Omron CX-Programmer project NewProject (CX-Programmer 9.73)

# PLC NewPLC1: CP1E N30

## Global symbols (name address type ; comment)
0.00 BOOL  ; START
0.01 BOOL  ; STOP
100.00 BOOL  ; LAMPU HIJAU SIMPANG 1
100.01 BOOL  ; LAMPU KUNING SIMPANG 1
100.02 BOOL  ; LAMPU MERAH SIMPANG 1
100.03 BOOL  ; LAMPU HIJAU SIMPANG 2
100.04 BOOL  ; LAMPU KUNING SIMPANG 2
100.05 BOOL  ; LAMPU MERAH SIMPANG 2
100.06 BOOL  ; LAMPU HIJAU SIMPANG 3
100.07 BOOL  ; LAMPU KUNING SIMPANG 3
100.08 BOOL  ; LAMPU MERAH SIMPANG 3
100.09 BOOL  ; LAMPU HIJAU SIMPANG 4
100.10 BOOL  ; LAMPU KUNING SIMPANG 4
100.11 BOOL  ; LAMPU MERAH SIMPANG 4
T000 BOOL  ; Tunggu Hijau 1
T001 BOOL  ; Tunggu Kuning 1
T002 BOOL  ; Tunggu Hijau 2
T003 BOOL  ; Tunggu Kuning 2
T004 BOOL  ; Tunggu Hijau 3
T005 BOOL  ; Tunggu Kuning 3
T006 BOOL  ; Tunggu Hijau 4
T007 BOOL  ; Tunggu Kuning 4
W0.00 BOOL  ; RUNNING

## Program NewProgram1 (cyclic task 0)

### Section Section1

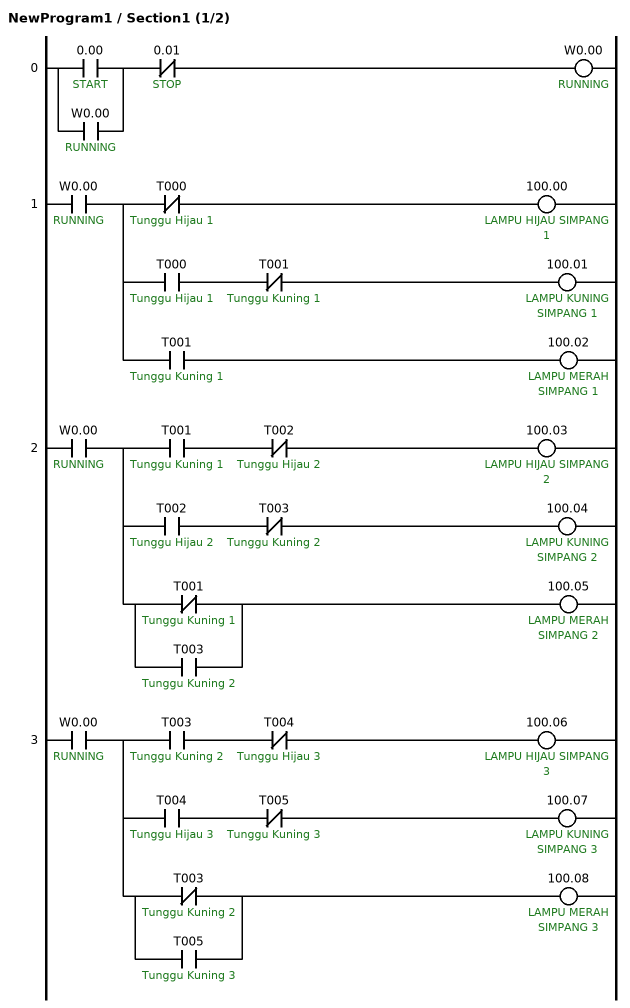
; rung 0
LD 0.00  ; START
OR W0.00  ; RUNNING
ANDNOT 0.01  ; STOP
OUT W0.00  ; RUNNING
; rung 1
LD W0.00  ; RUNNING
OUT TR0
ANDNOT T000  ; Tunggu Hijau 1
OUT 100.00  ; LAMPU HIJAU SIMPANG 1
LD TR0
AND T000  ; Tunggu Hijau 1
ANDNOT T001  ; Tunggu Kuning 1
OUT 100.01  ; LAMPU KUNING SIMPANG 1
LD TR0
AND T001  ; Tunggu Kuning 1
OUT 100.02  ; LAMPU MERAH SIMPANG 1
; rung 2
LD W0.00  ; RUNNING
OUT TR0
AND T001  ; Tunggu Kuning 1
ANDNOT T002  ; Tunggu Hijau 2
OUT 100.03  ; LAMPU HIJAU SIMPANG 2
LD TR0
AND T002  ; Tunggu Hijau 2
ANDNOT T003  ; Tunggu Kuning 2
OUT 100.04  ; LAMPU KUNING SIMPANG 2
LD TR0
LDNOT T001  ; Tunggu Kuning 1
OR T003  ; Tunggu Kuning 2
ANDLD
OUT 100.05  ; LAMPU MERAH SIMPANG 2
; rung 3
LD W0.00  ; RUNNING
OUT TR0
AND T003  ; Tunggu Kuning 2
ANDNOT T004  ; Tunggu Hijau 3
OUT 100.06  ; LAMPU HIJAU SIMPANG 3
LD TR0
AND T004  ; Tunggu Hijau 3
ANDNOT T005  ; Tunggu Kuning 3
OUT 100.07  ; LAMPU KUNING SIMPANG 3
LD TR0
LDNOT T003  ; Tunggu Kuning 2
OR T005  ; Tunggu Kuning 3
ANDLD
OUT 100.08  ; LAMPU MERAH SIMPANG 3

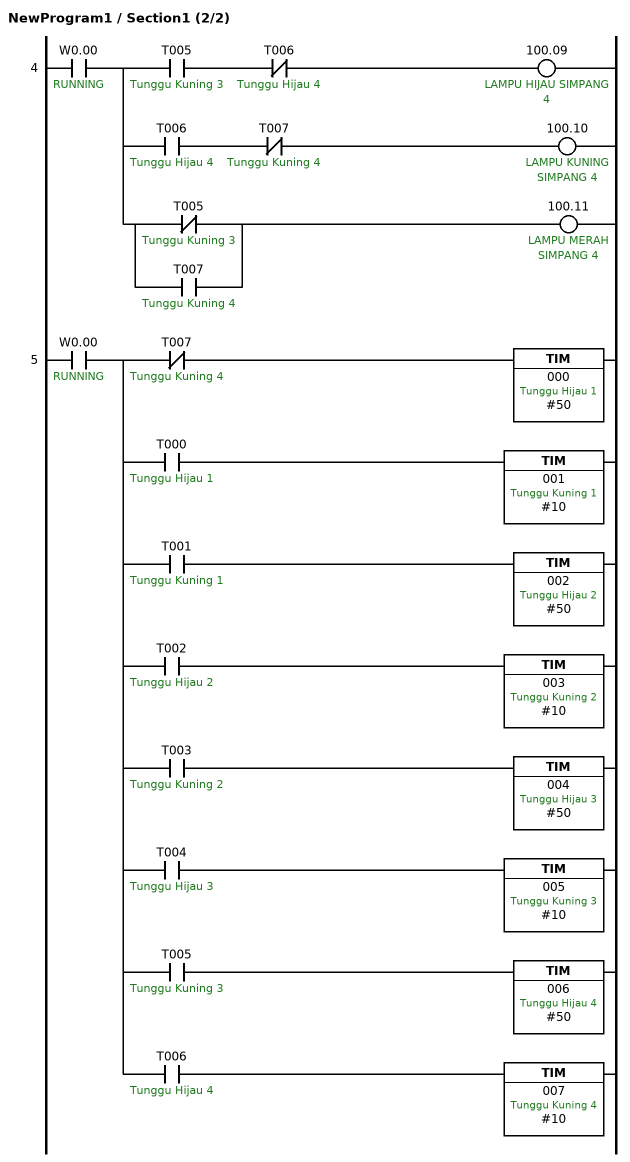
; rung 4
LD W0.00  ; RUNNING
OUT TR0
AND T005  ; Tunggu Kuning 3
ANDNOT T006  ; Tunggu Hijau 4
OUT 100.09  ; LAMPU HIJAU SIMPANG 4
LD TR0
AND T006  ; Tunggu Hijau 4
ANDNOT T007  ; Tunggu Kuning 4
OUT 100.10  ; LAMPU KUNING SIMPANG 4
LD TR0
LDNOT T005  ; Tunggu Kuning 3
OR T007  ; Tunggu Kuning 4
ANDLD
OUT 100.11  ; LAMPU MERAH SIMPANG 4
; rung 5
LD W0.00  ; RUNNING
OUT TR0
ANDNOT T007  ; Tunggu Kuning 4
TIM 000 #50  ; Tunggu Hijau 1
LD TR0
AND T000  ; Tunggu Hijau 1
TIM 001 #10  ; Tunggu Kuning 1
LD TR0
AND T001  ; Tunggu Kuning 1
TIM 002 #50  ; Tunggu Hijau 2
LD TR0
AND T002  ; Tunggu Hijau 2
TIM 003 #10  ; Tunggu Kuning 2
LD TR0
AND T003  ; Tunggu Kuning 2
TIM 004 #50  ; Tunggu Hijau 3
LD TR0
AND T004  ; Tunggu Hijau 3
TIM 005 #10  ; Tunggu Kuning 3
LD TR0
AND T005  ; Tunggu Kuning 3
TIM 006 #50  ; Tunggu Hijau 4
LD TR0
AND T006  ; Tunggu Hijau 4
TIM 007 #10  ; Tunggu Kuning 4

### Section END
; rung 0
END(001)